// TIA Portal V15.1 export
// export: Created 2024-05-17T05:38:57.2674434Z, ExportSetting WithDefaults, DisplayName Totally Integrated Automation Portal, DisplayVersion V15.1 Update 5, DisplayName TIA Portal Openness, DisplayVersion V15.1 Update 5, DisplayName SINAMICS Startdrive Advanced, DisplayVersion V15.1, DisplayName G130, G150, S120, S150, SINAMICS MV, S210, DisplayVersion V15.1, DisplayName G110M, G120, G120C, G120D, G120P, DisplayVersion V15.1, DisplayName STEP 7 Professional, DisplayVersion V15.1 Update 5, DisplayName STEP 7 Safety, DisplayVersion V15.1, DisplayName WinCC Professional, DisplayVersion V15.1 Update 5, DisplayName SIMATIC Visualization Architect, DisplayVersion V15.1
FUNCTION "209210ZS01PNIODiag" : Void   // FC324, FBD
TITLE = 209210ZS01PNIODiag
{ S7_Optimized_Access := 'FALSE' }
AUTHOR : JS
NAME : Mot001
VERSION : 0.1
// stored: AutoNumber false, IsIECCheckEnabled false, SetENOAutomatically False, UDAEnableTagReadback false
   VAR_OUTPUT
      O_AlarmA : Bool;   // Alarm A
      O_AlarmB : Bool;   // Alarm B
      O_AlarmC : Bool;   // Alarm C
      O_AlarmD : Bool;   // Alarm D
      O_AlarmABCondition : Bool;   // Alarms resetable
      H_IAnim : Word;   // Animation bits to Icon in WinCC
   END_VAR
   VAR_TEMP   // added for the SCL form of the ladder/FBD networks
      _w1 : Bool;
   END_VAR
BEGIN

REGION Network 1: **** --------------------- ET200sp I/O --------------------- ****
END_REGION

REGION Network 2: **** 3 - Communication - Devices **** 209210AS10-JW40 - ET200sp I/O - Busnode 210AS10 - node 40
   // Profinet device don't exist - ET200sp I/O - Busnode 210AS10 - node 40
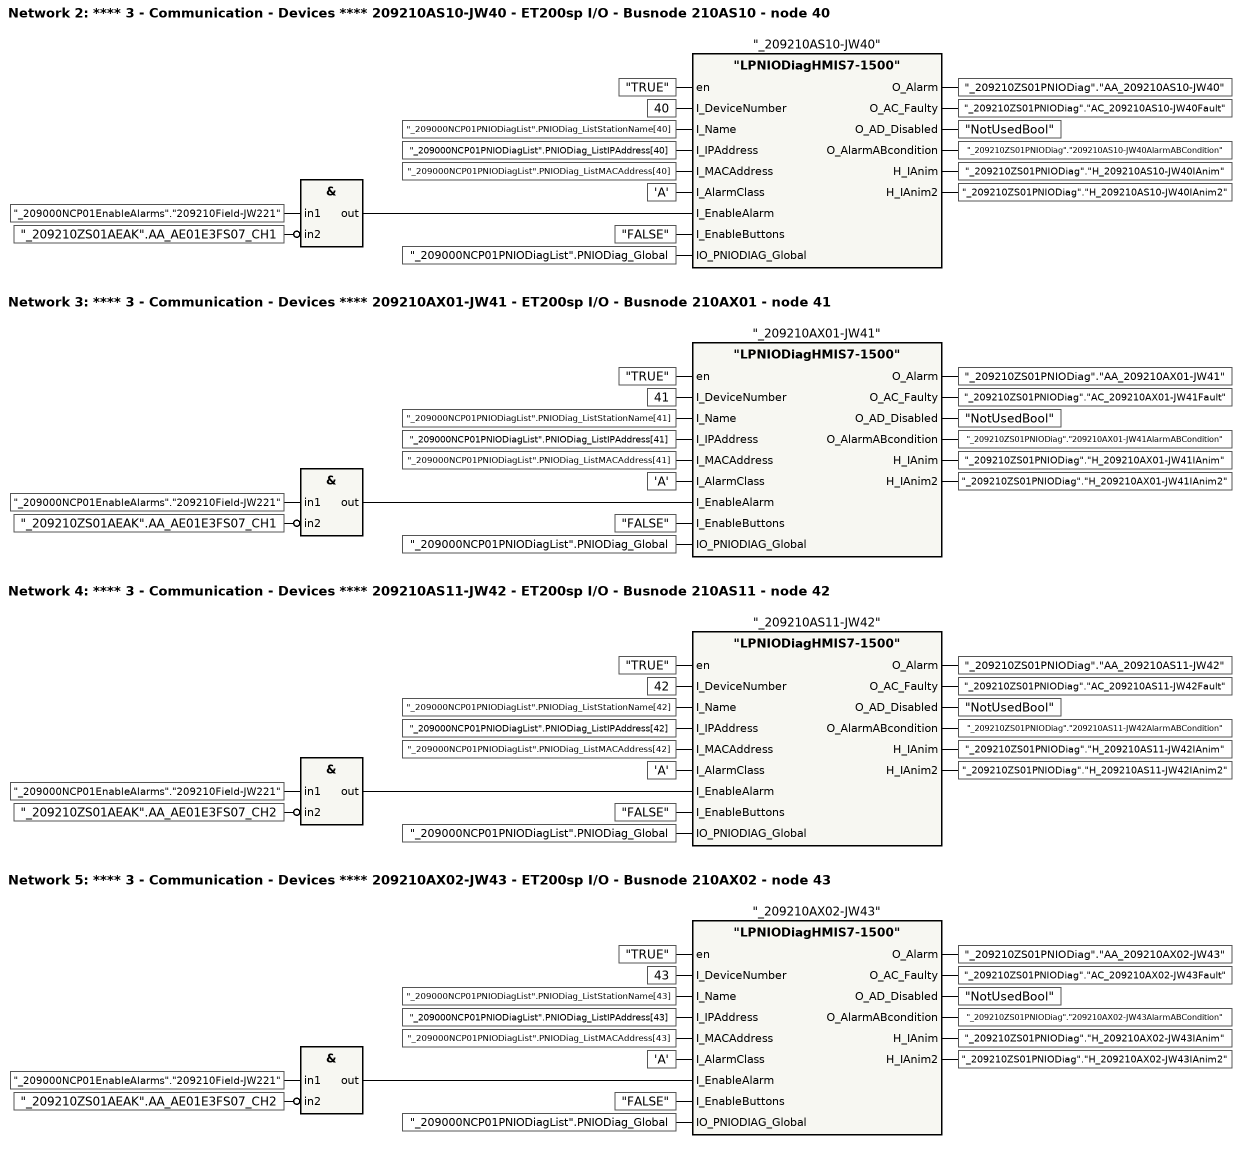
   IF "TRUE" THEN
       "_209210AS10-JW40"(I_DeviceNumber := 40,   // "LPNIODiagHMIS7-1500"
                          I_Name := "_209000NCP01PNIODiagList".PNIODiag_ListStationName[40],
                          I_IPAddress := "_209000NCP01PNIODiagList".PNIODiag_ListIPAddress[40],
                          I_MACAddress := "_209000NCP01PNIODiagList".PNIODiag_ListMACAddress[40],
                          I_AlarmClass := 'A',
                          I_EnableAlarm := "_209000NCP01EnableAlarms"."209210Field-JW221" AND NOT "_209210ZS01AEAK".AA_AE01E3FS07_CH1,
                          I_EnableButtons := "FALSE",
                          IO_PNIODIAG_Global := "_209000NCP01PNIODiagList".PNIODiag_Global,
                          O_Alarm => "_209210ZS01PNIODiag"."AA_209210AS10-JW40",
                          O_AC_Faulty => "_209210ZS01PNIODiag"."AC_209210AS10-JW40Fault",
                          O_AD_Disabled => "NotUsedBool",
                          O_AlarmABcondition => "_209210ZS01PNIODiag"."209210AS10-JW40AlarmABCondition",
                          H_IAnim => "_209210ZS01PNIODiag"."H_209210AS10-JW40IAnim",
                          H_IAnim2 => "_209210ZS01PNIODiag"."H_209210AS10-JW40IAnim2");
   END_IF;
END_REGION

REGION Network 3: **** 3 - Communication - Devices **** 209210AX01-JW41 - ET200sp I/O - Busnode 210AX01 - node 41
   // Profinet device don't exist - ET200sp I/O - Busnode 210AX01 - node 41
   IF "TRUE" THEN
       "_209210AX01-JW41"(I_DeviceNumber := 41,   // "LPNIODiagHMIS7-1500"
                          I_Name := "_209000NCP01PNIODiagList".PNIODiag_ListStationName[41],
                          I_IPAddress := "_209000NCP01PNIODiagList".PNIODiag_ListIPAddress[41],
                          I_MACAddress := "_209000NCP01PNIODiagList".PNIODiag_ListMACAddress[41],
                          I_AlarmClass := 'A',
                          I_EnableAlarm := "_209000NCP01EnableAlarms"."209210Field-JW221" AND NOT "_209210ZS01AEAK".AA_AE01E3FS07_CH1,
                          I_EnableButtons := "FALSE",
                          IO_PNIODIAG_Global := "_209000NCP01PNIODiagList".PNIODiag_Global,
                          O_Alarm => "_209210ZS01PNIODiag"."AA_209210AX01-JW41",
                          O_AC_Faulty => "_209210ZS01PNIODiag"."AC_209210AX01-JW41Fault",
                          O_AD_Disabled => "NotUsedBool",
                          O_AlarmABcondition => "_209210ZS01PNIODiag"."209210AX01-JW41AlarmABCondition",
                          H_IAnim => "_209210ZS01PNIODiag"."H_209210AX01-JW41IAnim",
                          H_IAnim2 => "_209210ZS01PNIODiag"."H_209210AX01-JW41IAnim2");
   END_IF;
END_REGION

REGION Network 4: **** 3 - Communication - Devices **** 209210AS11-JW42 - ET200sp I/O - Busnode 210AS11 - node 42
   // Profinet device don't exist - ET200sp I/O - Busnode 210AS11 - node 42
   IF "TRUE" THEN
       "_209210AS11-JW42"(I_DeviceNumber := 42,   // "LPNIODiagHMIS7-1500"
                          I_Name := "_209000NCP01PNIODiagList".PNIODiag_ListStationName[42],
                          I_IPAddress := "_209000NCP01PNIODiagList".PNIODiag_ListIPAddress[42],
                          I_MACAddress := "_209000NCP01PNIODiagList".PNIODiag_ListMACAddress[42],
                          I_AlarmClass := 'A',
                          I_EnableAlarm := "_209000NCP01EnableAlarms"."209210Field-JW221" AND NOT "_209210ZS01AEAK".AA_AE01E3FS07_CH2,
                          I_EnableButtons := "FALSE",
                          IO_PNIODIAG_Global := "_209000NCP01PNIODiagList".PNIODiag_Global,
                          O_Alarm => "_209210ZS01PNIODiag"."AA_209210AS11-JW42",
                          O_AC_Faulty => "_209210ZS01PNIODiag"."AC_209210AS11-JW42Fault",
                          O_AD_Disabled => "NotUsedBool",
                          O_AlarmABcondition => "_209210ZS01PNIODiag"."209210AS11-JW42AlarmABCondition",
                          H_IAnim => "_209210ZS01PNIODiag"."H_209210AS11-JW42IAnim",
                          H_IAnim2 => "_209210ZS01PNIODiag"."H_209210AS11-JW42IAnim2");
   END_IF;
END_REGION

REGION Network 5: **** 3 - Communication - Devices **** 209210AX02-JW43 - ET200sp I/O - Busnode 210AX02 - node 43
   // Profinet device don't exist - ET200sp I/O - Busnode 210AX02 - node 43
   IF "TRUE" THEN
       "_209210AX02-JW43"(I_DeviceNumber := 43,   // "LPNIODiagHMIS7-1500"
                          I_Name := "_209000NCP01PNIODiagList".PNIODiag_ListStationName[43],
                          I_IPAddress := "_209000NCP01PNIODiagList".PNIODiag_ListIPAddress[43],
                          I_MACAddress := "_209000NCP01PNIODiagList".PNIODiag_ListMACAddress[43],
                          I_AlarmClass := 'A',
                          I_EnableAlarm := "_209000NCP01EnableAlarms"."209210Field-JW221" AND NOT "_209210ZS01AEAK".AA_AE01E3FS07_CH2,
                          I_EnableButtons := "FALSE",
                          IO_PNIODIAG_Global := "_209000NCP01PNIODiagList".PNIODiag_Global,
                          O_Alarm => "_209210ZS01PNIODiag"."AA_209210AX02-JW43",
                          O_AC_Faulty => "_209210ZS01PNIODiag"."AC_209210AX02-JW43Fault",
                          O_AD_Disabled => "NotUsedBool",
                          O_AlarmABcondition => "_209210ZS01PNIODiag"."209210AX02-JW43AlarmABCondition",
                          H_IAnim => "_209210ZS01PNIODiag"."H_209210AX02-JW43IAnim",
                          H_IAnim2 => "_209210ZS01PNIODiag"."H_209210AX02-JW43IAnim2");
   END_IF;
END_REGION

REGION Network 6: **** 3 - Communication - Devices **** 209210AS20-JW48 - ET200sp I/O - Busnode 210AS20 - node 48
   // Profinet device don't exist - ET200sp I/O - Busnode 210AS20 - node 48
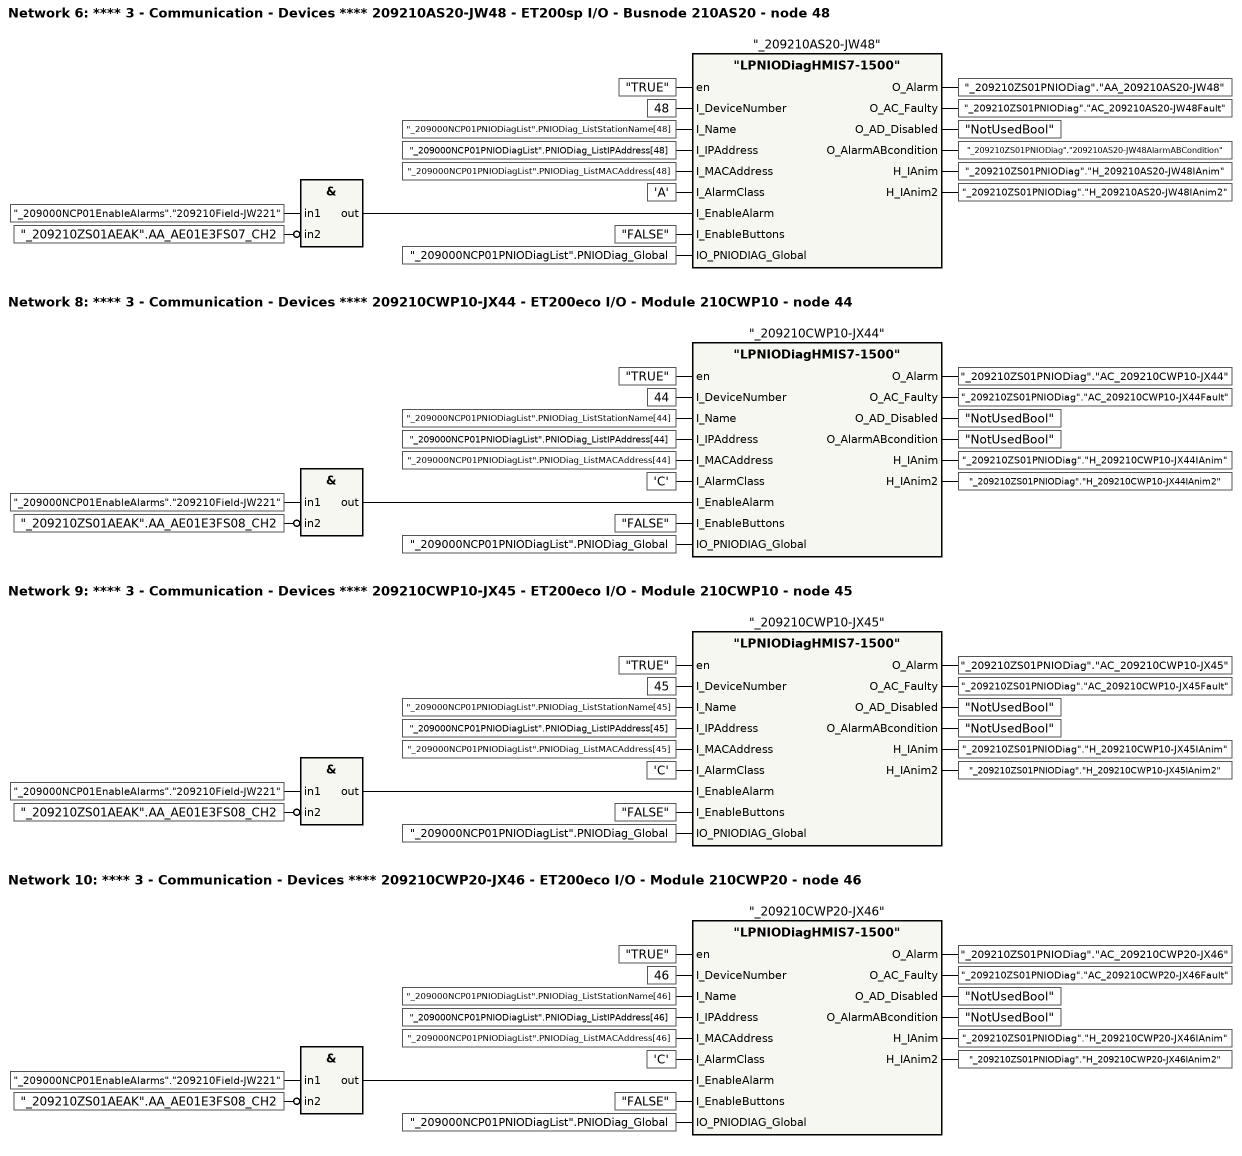
   IF "TRUE" THEN
       "_209210AS20-JW48"(I_DeviceNumber := 48,   // "LPNIODiagHMIS7-1500"
                          I_Name := "_209000NCP01PNIODiagList".PNIODiag_ListStationName[48],
                          I_IPAddress := "_209000NCP01PNIODiagList".PNIODiag_ListIPAddress[48],
                          I_MACAddress := "_209000NCP01PNIODiagList".PNIODiag_ListMACAddress[48],
                          I_AlarmClass := 'A',
                          I_EnableAlarm := "_209000NCP01EnableAlarms"."209210Field-JW221" AND NOT "_209210ZS01AEAK".AA_AE01E3FS07_CH2,
                          I_EnableButtons := "FALSE",
                          IO_PNIODIAG_Global := "_209000NCP01PNIODiagList".PNIODiag_Global,
                          O_Alarm => "_209210ZS01PNIODiag"."AA_209210AS20-JW48",
                          O_AC_Faulty => "_209210ZS01PNIODiag"."AC_209210AS20-JW48Fault",
                          O_AD_Disabled => "NotUsedBool",
                          O_AlarmABcondition => "_209210ZS01PNIODiag"."209210AS20-JW48AlarmABCondition",
                          H_IAnim => "_209210ZS01PNIODiag"."H_209210AS20-JW48IAnim",
                          H_IAnim2 => "_209210ZS01PNIODiag"."H_209210AS20-JW48IAnim2");
   END_IF;
END_REGION

REGION Network 7: **** --------------------- ET200eco I/O --------------------- ****
END_REGION

REGION Network 8: **** 3 - Communication - Devices **** 209210CWP10-JX44 - ET200eco I/O - Module 210CWP10 - node 44
   // Profinet device don't exist - ET200eco I/O - Module 210CWP10 - node 44
   IF "TRUE" THEN
       "_209210CWP10-JX44"(I_DeviceNumber := 44,   // "LPNIODiagHMIS7-1500"
                           I_Name := "_209000NCP01PNIODiagList".PNIODiag_ListStationName[44],
                           I_IPAddress := "_209000NCP01PNIODiagList".PNIODiag_ListIPAddress[44],
                           I_MACAddress := "_209000NCP01PNIODiagList".PNIODiag_ListMACAddress[44],
                           I_AlarmClass := 'C',
                           I_EnableAlarm := "_209000NCP01EnableAlarms"."209210Field-JW221" AND NOT "_209210ZS01AEAK".AA_AE01E3FS08_CH2,
                           I_EnableButtons := "FALSE",
                           IO_PNIODIAG_Global := "_209000NCP01PNIODiagList".PNIODiag_Global,
                           O_Alarm => "_209210ZS01PNIODiag"."AC_209210CWP10-JX44",
                           O_AC_Faulty => "_209210ZS01PNIODiag"."AC_209210CWP10-JX44Fault",
                           O_AD_Disabled => "NotUsedBool",
                           O_AlarmABcondition => "NotUsedBool",
                           H_IAnim => "_209210ZS01PNIODiag"."H_209210CWP10-JX44IAnim",
                           H_IAnim2 => "_209210ZS01PNIODiag"."H_209210CWP10-JX44IAnim2");
   END_IF;
END_REGION

REGION Network 9: **** 3 - Communication - Devices **** 209210CWP10-JX45 - ET200eco I/O - Module 210CWP10 - node 45
   // Profinet device don't exist - ET200eco I/O - Module 210CWP10 - node 45
   IF "TRUE" THEN
       "_209210CWP10-JX45"(I_DeviceNumber := 45,   // "LPNIODiagHMIS7-1500"
                           I_Name := "_209000NCP01PNIODiagList".PNIODiag_ListStationName[45],
                           I_IPAddress := "_209000NCP01PNIODiagList".PNIODiag_ListIPAddress[45],
                           I_MACAddress := "_209000NCP01PNIODiagList".PNIODiag_ListMACAddress[45],
                           I_AlarmClass := 'C',
                           I_EnableAlarm := "_209000NCP01EnableAlarms"."209210Field-JW221" AND NOT "_209210ZS01AEAK".AA_AE01E3FS08_CH2,
                           I_EnableButtons := "FALSE",
                           IO_PNIODIAG_Global := "_209000NCP01PNIODiagList".PNIODiag_Global,
                           O_Alarm => "_209210ZS01PNIODiag"."AC_209210CWP10-JX45",
                           O_AC_Faulty => "_209210ZS01PNIODiag"."AC_209210CWP10-JX45Fault",
                           O_AD_Disabled => "NotUsedBool",
                           O_AlarmABcondition => "NotUsedBool",
                           H_IAnim => "_209210ZS01PNIODiag"."H_209210CWP10-JX45IAnim",
                           H_IAnim2 => "_209210ZS01PNIODiag"."H_209210CWP10-JX45IAnim2");
   END_IF;
END_REGION

REGION Network 10: **** 3 - Communication - Devices **** 209210CWP20-JX46 - ET200eco I/O - Module 210CWP20 - node 46
   // Profinet device don't exist - ET200eco I/O - Module 210CWP20 - node 46
   IF "TRUE" THEN
       "_209210CWP20-JX46"(I_DeviceNumber := 46,   // "LPNIODiagHMIS7-1500"
                           I_Name := "_209000NCP01PNIODiagList".PNIODiag_ListStationName[46],
                           I_IPAddress := "_209000NCP01PNIODiagList".PNIODiag_ListIPAddress[46],
                           I_MACAddress := "_209000NCP01PNIODiagList".PNIODiag_ListMACAddress[46],
                           I_AlarmClass := 'C',
                           I_EnableAlarm := "_209000NCP01EnableAlarms"."209210Field-JW221" AND NOT "_209210ZS01AEAK".AA_AE01E3FS08_CH2,
                           I_EnableButtons := "FALSE",
                           IO_PNIODIAG_Global := "_209000NCP01PNIODiagList".PNIODiag_Global,
                           O_Alarm => "_209210ZS01PNIODiag"."AC_209210CWP20-JX46",
                           O_AC_Faulty => "_209210ZS01PNIODiag"."AC_209210CWP20-JX46Fault",
                           O_AD_Disabled => "NotUsedBool",
                           O_AlarmABcondition => "NotUsedBool",
                           H_IAnim => "_209210ZS01PNIODiag"."H_209210CWP20-JX46IAnim",
                           H_IAnim2 => "_209210ZS01PNIODiag"."H_209210CWP20-JX46IAnim2");
   END_IF;
END_REGION

REGION Network 11: **** 3 - Communication - Devices **** 209210CWP20-JX47 - ET200eco I/O - Module 210CWP20 - node 47
   // Profinet device don't exist - ET200eco I/O - Module 210CWP20 - node 47
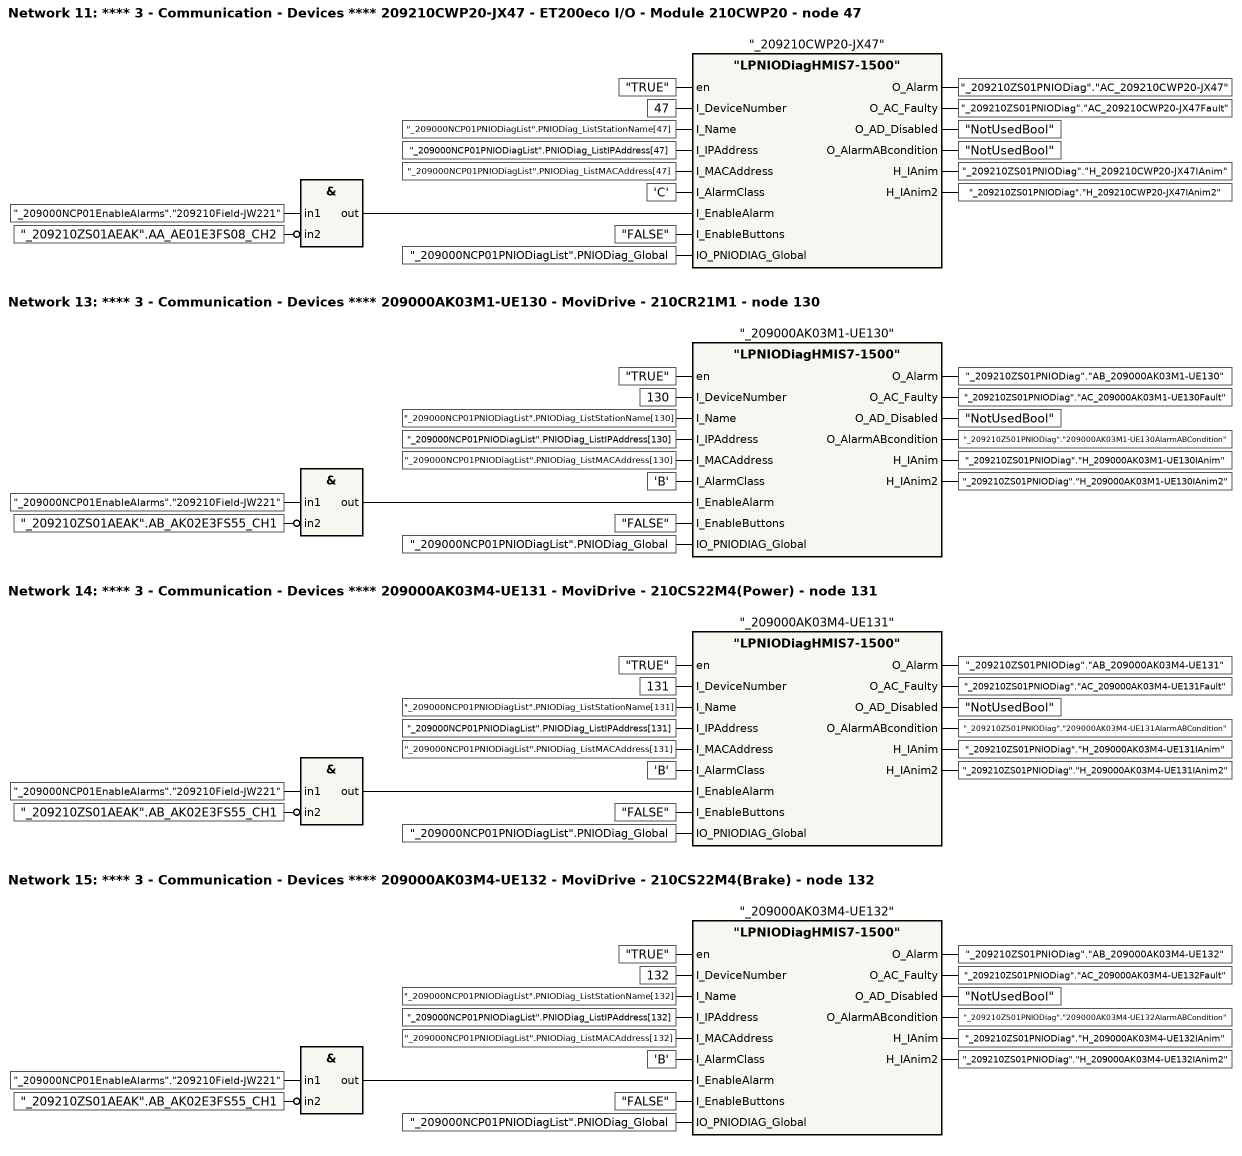
   IF "TRUE" THEN
       "_209210CWP20-JX47"(I_DeviceNumber := 47,   // "LPNIODiagHMIS7-1500"
                           I_Name := "_209000NCP01PNIODiagList".PNIODiag_ListStationName[47],
                           I_IPAddress := "_209000NCP01PNIODiagList".PNIODiag_ListIPAddress[47],
                           I_MACAddress := "_209000NCP01PNIODiagList".PNIODiag_ListMACAddress[47],
                           I_AlarmClass := 'C',
                           I_EnableAlarm := "_209000NCP01EnableAlarms"."209210Field-JW221" AND NOT "_209210ZS01AEAK".AA_AE01E3FS08_CH2,
                           I_EnableButtons := "FALSE",
                           IO_PNIODIAG_Global := "_209000NCP01PNIODiagList".PNIODiag_Global,
                           O_Alarm => "_209210ZS01PNIODiag"."AC_209210CWP20-JX47",
                           O_AC_Faulty => "_209210ZS01PNIODiag"."AC_209210CWP20-JX47Fault",
                           O_AD_Disabled => "NotUsedBool",
                           O_AlarmABcondition => "NotUsedBool",
                           H_IAnim => "_209210ZS01PNIODiag"."H_209210CWP20-JX47IAnim",
                           H_IAnim2 => "_209210ZS01PNIODiag"."H_209210CWP20-JX47IAnim2");
   END_IF;
END_REGION

REGION Network 12: **** --------------------- Drive --------------------- ****
END_REGION

REGION Network 13: **** 3 - Communication - Devices **** 209000AK03M1-UE130 - MoviDrive - 210CR21M1 - node 130
   // Profinet device don't exist - MoviDrive - 210CR21M1 - node 130
   IF "TRUE" THEN
       "_209000AK03M1-UE130"(I_DeviceNumber := 130,   // "LPNIODiagHMIS7-1500"
                             I_Name := "_209000NCP01PNIODiagList".PNIODiag_ListStationName[130],
                             I_IPAddress := "_209000NCP01PNIODiagList".PNIODiag_ListIPAddress[130],
                             I_MACAddress := "_209000NCP01PNIODiagList".PNIODiag_ListMACAddress[130],
                             I_AlarmClass := 'B',
                             I_EnableAlarm := "_209000NCP01EnableAlarms"."209210Field-JW221" AND NOT "_209210ZS01AEAK".AB_AK02E3FS55_CH1,
                             I_EnableButtons := "FALSE",
                             IO_PNIODIAG_Global := "_209000NCP01PNIODiagList".PNIODiag_Global,
                             O_Alarm => "_209210ZS01PNIODiag"."AB_209000AK03M1-UE130",
                             O_AC_Faulty => "_209210ZS01PNIODiag"."AC_209000AK03M1-UE130Fault",
                             O_AD_Disabled => "NotUsedBool",
                             O_AlarmABcondition => "_209210ZS01PNIODiag"."209000AK03M1-UE130AlarmABCondition",
                             H_IAnim => "_209210ZS01PNIODiag"."H_209000AK03M1-UE130IAnim",
                             H_IAnim2 => "_209210ZS01PNIODiag"."H_209000AK03M1-UE130IAnim2");
   END_IF;
END_REGION

REGION Network 14: **** 3 - Communication - Devices **** 209000AK03M4-UE131 - MoviDrive - 210CS22M4(Power) - node 131
   // Profinet device don't exist - MoviDrive - 210CS22M4(Power) - node 131
   IF "TRUE" THEN
       "_209000AK03M4-UE131"(I_DeviceNumber := 131,   // "LPNIODiagHMIS7-1500"
                             I_Name := "_209000NCP01PNIODiagList".PNIODiag_ListStationName[131],
                             I_IPAddress := "_209000NCP01PNIODiagList".PNIODiag_ListIPAddress[131],
                             I_MACAddress := "_209000NCP01PNIODiagList".PNIODiag_ListMACAddress[131],
                             I_AlarmClass := 'B',
                             I_EnableAlarm := "_209000NCP01EnableAlarms"."209210Field-JW221" AND NOT "_209210ZS01AEAK".AB_AK02E3FS55_CH1,
                             I_EnableButtons := "FALSE",
                             IO_PNIODIAG_Global := "_209000NCP01PNIODiagList".PNIODiag_Global,
                             O_Alarm => "_209210ZS01PNIODiag"."AB_209000AK03M4-UE131",
                             O_AC_Faulty => "_209210ZS01PNIODiag"."AC_209000AK03M4-UE131Fault",
                             O_AD_Disabled => "NotUsedBool",
                             O_AlarmABcondition => "_209210ZS01PNIODiag"."209000AK03M4-UE131AlarmABCondition",
                             H_IAnim => "_209210ZS01PNIODiag"."H_209000AK03M4-UE131IAnim",
                             H_IAnim2 => "_209210ZS01PNIODiag"."H_209000AK03M4-UE131IAnim2");
   END_IF;
END_REGION

REGION Network 15: **** 3 - Communication - Devices **** 209000AK03M4-UE132 - MoviDrive - 210CS22M4(Brake) - node 132
   // Profinet device don't exist - MoviDrive - 210CS22M4(Brake) - node 132
   IF "TRUE" THEN
       "_209000AK03M4-UE132"(I_DeviceNumber := 132,   // "LPNIODiagHMIS7-1500"
                             I_Name := "_209000NCP01PNIODiagList".PNIODiag_ListStationName[132],
                             I_IPAddress := "_209000NCP01PNIODiagList".PNIODiag_ListIPAddress[132],
                             I_MACAddress := "_209000NCP01PNIODiagList".PNIODiag_ListMACAddress[132],
                             I_AlarmClass := 'B',
                             I_EnableAlarm := "_209000NCP01EnableAlarms"."209210Field-JW221" AND NOT "_209210ZS01AEAK".AB_AK02E3FS55_CH1,
                             I_EnableButtons := "FALSE",
                             IO_PNIODIAG_Global := "_209000NCP01PNIODiagList".PNIODiag_Global,
                             O_Alarm => "_209210ZS01PNIODiag"."AB_209000AK03M4-UE132",
                             O_AC_Faulty => "_209210ZS01PNIODiag"."AC_209000AK03M4-UE132Fault",
                             O_AD_Disabled => "NotUsedBool",
                             O_AlarmABcondition => "_209210ZS01PNIODiag"."209000AK03M4-UE132AlarmABCondition",
                             H_IAnim => "_209210ZS01PNIODiag"."H_209000AK03M4-UE132IAnim",
                             H_IAnim2 => "_209210ZS01PNIODiag"."H_209000AK03M4-UE132IAnim2");
   END_IF;
END_REGION

REGION Network 16: **** 3 - Communication - Devices **** 209000AK03M1-UE133 - MoviDrive - 210CR23M1 - node 133
   // Profinet device don't exist - MoviDrive - 210CR23M1 - node 133
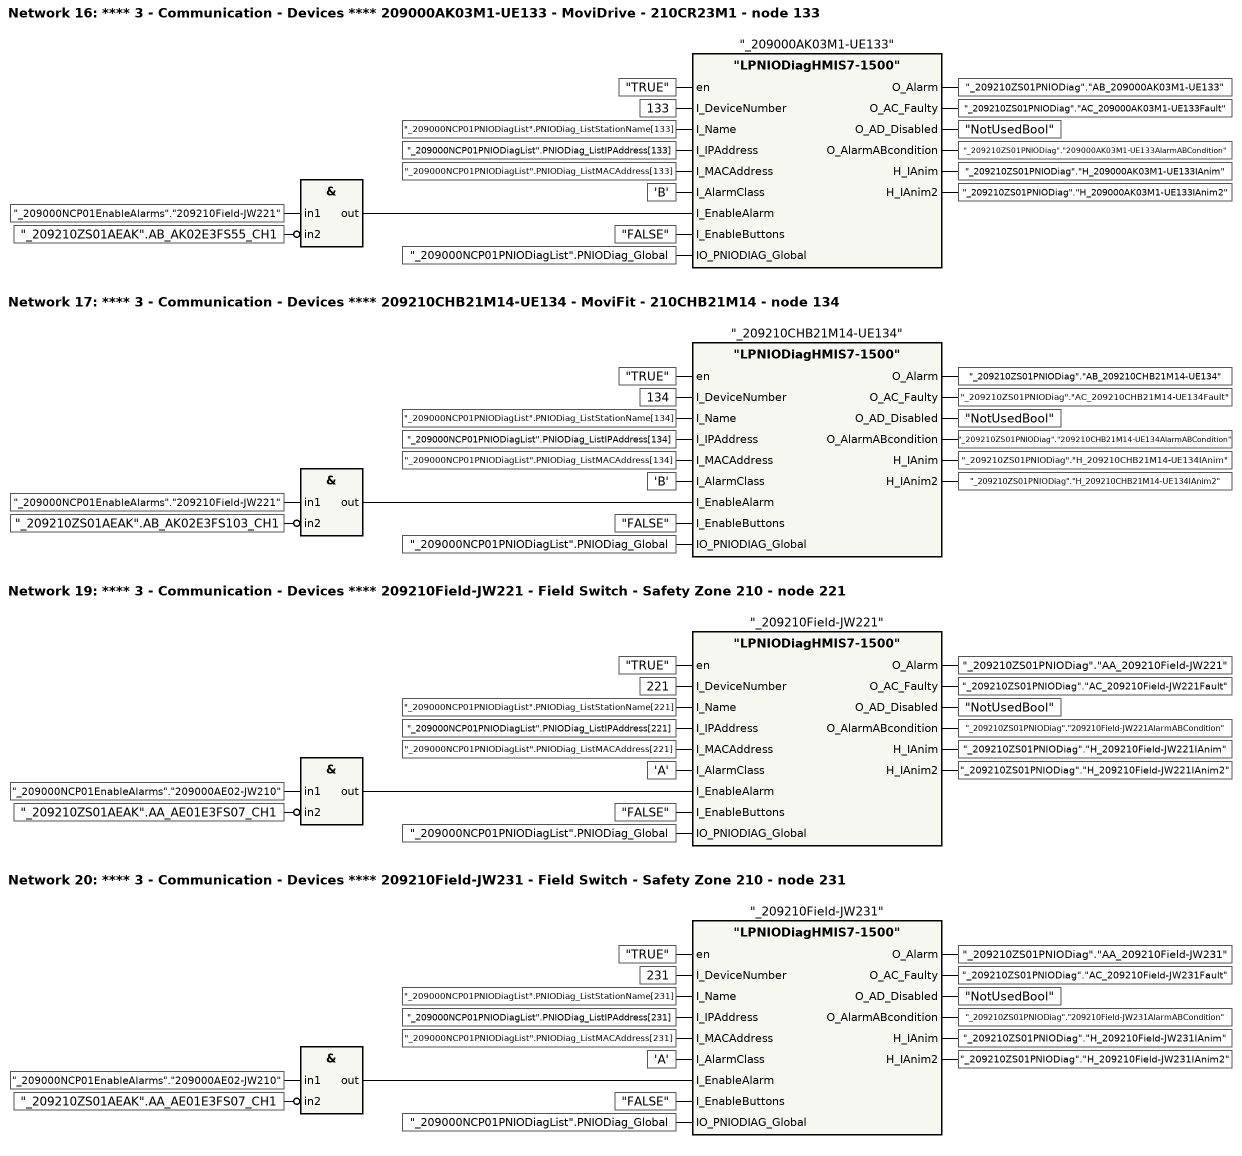
   IF "TRUE" THEN
       "_209000AK03M1-UE133"(I_DeviceNumber := 133,   // "LPNIODiagHMIS7-1500"
                             I_Name := "_209000NCP01PNIODiagList".PNIODiag_ListStationName[133],
                             I_IPAddress := "_209000NCP01PNIODiagList".PNIODiag_ListIPAddress[133],
                             I_MACAddress := "_209000NCP01PNIODiagList".PNIODiag_ListMACAddress[133],
                             I_AlarmClass := 'B',
                             I_EnableAlarm := "_209000NCP01EnableAlarms"."209210Field-JW221" AND NOT "_209210ZS01AEAK".AB_AK02E3FS55_CH1,
                             I_EnableButtons := "FALSE",
                             IO_PNIODIAG_Global := "_209000NCP01PNIODiagList".PNIODiag_Global,
                             O_Alarm => "_209210ZS01PNIODiag"."AB_209000AK03M1-UE133",
                             O_AC_Faulty => "_209210ZS01PNIODiag"."AC_209000AK03M1-UE133Fault",
                             O_AD_Disabled => "NotUsedBool",
                             O_AlarmABcondition => "_209210ZS01PNIODiag"."209000AK03M1-UE133AlarmABCondition",
                             H_IAnim => "_209210ZS01PNIODiag"."H_209000AK03M1-UE133IAnim",
                             H_IAnim2 => "_209210ZS01PNIODiag"."H_209000AK03M1-UE133IAnim2");
   END_IF;
END_REGION

REGION Network 17: **** 3 - Communication - Devices **** 209210CHB21M14-UE134 - MoviFit - 210CHB21M14 - node 134
   // Profinet device don't exist - MoviFit - 210CHB21M14 - node 134
   IF "TRUE" THEN
       "_209210CHB21M14-UE134"(I_DeviceNumber := 134,   // "LPNIODiagHMIS7-1500"
                               I_Name := "_209000NCP01PNIODiagList".PNIODiag_ListStationName[134],
                               I_IPAddress := "_209000NCP01PNIODiagList".PNIODiag_ListIPAddress[134],
                               I_MACAddress := "_209000NCP01PNIODiagList".PNIODiag_ListMACAddress[134],
                               I_AlarmClass := 'B',
                               I_EnableAlarm := "_209000NCP01EnableAlarms"."209210Field-JW221" AND NOT "_209210ZS01AEAK".AB_AK02E3FS103_CH1,
                               I_EnableButtons := "FALSE",
                               IO_PNIODIAG_Global := "_209000NCP01PNIODiagList".PNIODiag_Global,
                               O_Alarm => "_209210ZS01PNIODiag"."AB_209210CHB21M14-UE134",
                               O_AC_Faulty => "_209210ZS01PNIODiag"."AC_209210CHB21M14-UE134Fault",
                               O_AD_Disabled => "NotUsedBool",
                               O_AlarmABcondition => "_209210ZS01PNIODiag"."209210CHB21M14-UE134AlarmABCondition",
                               H_IAnim => "_209210ZS01PNIODiag"."H_209210CHB21M14-UE134IAnim",
                               H_IAnim2 => "_209210ZS01PNIODiag"."H_209210CHB21M14-UE134IAnim2");
   END_IF;
END_REGION

REGION Network 18: **** --------------------- Field Switch --------------------- ****
END_REGION

REGION Network 19: **** 3 - Communication - Devices **** 209210Field-JW221 - Field Switch - Safety Zone 210 - node 221
   // Profinet device don't exist - Field Switch - Safety Zone 210 - node 221
   IF "TRUE" THEN
       "_209210Field-JW221"(I_DeviceNumber := 221,   // "LPNIODiagHMIS7-1500"
                            I_Name := "_209000NCP01PNIODiagList".PNIODiag_ListStationName[221],
                            I_IPAddress := "_209000NCP01PNIODiagList".PNIODiag_ListIPAddress[221],
                            I_MACAddress := "_209000NCP01PNIODiagList".PNIODiag_ListMACAddress[221],
                            I_AlarmClass := 'A',
                            I_EnableAlarm := "_209000NCP01EnableAlarms"."209000AE02-JW210" AND NOT "_209210ZS01AEAK".AA_AE01E3FS07_CH1,
                            I_EnableButtons := "FALSE",
                            IO_PNIODIAG_Global := "_209000NCP01PNIODiagList".PNIODiag_Global,
                            O_Alarm => "_209210ZS01PNIODiag"."AA_209210Field-JW221",
                            O_AC_Faulty => "_209210ZS01PNIODiag"."AC_209210Field-JW221Fault",
                            O_AD_Disabled => "NotUsedBool",
                            O_AlarmABcondition => "_209210ZS01PNIODiag"."209210Field-JW221AlarmABCondition",
                            H_IAnim => "_209210ZS01PNIODiag"."H_209210Field-JW221IAnim",
                            H_IAnim2 => "_209210ZS01PNIODiag"."H_209210Field-JW221IAnim2");
   END_IF;
END_REGION

REGION Network 20: **** 3 - Communication - Devices **** 209210Field-JW231 - Field Switch - Safety Zone 210 - node 231
   // Profinet device don't exist - Field Switch - Safety Zone 210 - node 231
   IF "TRUE" THEN
       "_209210Field-JW231"(I_DeviceNumber := 231,   // "LPNIODiagHMIS7-1500"
                            I_Name := "_209000NCP01PNIODiagList".PNIODiag_ListStationName[231],
                            I_IPAddress := "_209000NCP01PNIODiagList".PNIODiag_ListIPAddress[231],
                            I_MACAddress := "_209000NCP01PNIODiagList".PNIODiag_ListMACAddress[231],
                            I_AlarmClass := 'A',
                            I_EnableAlarm := "_209000NCP01EnableAlarms"."209000AE02-JW210" AND NOT "_209210ZS01AEAK".AA_AE01E3FS07_CH1,
                            I_EnableButtons := "FALSE",
                            IO_PNIODIAG_Global := "_209000NCP01PNIODiagList".PNIODiag_Global,
                            O_Alarm => "_209210ZS01PNIODiag"."AA_209210Field-JW231",
                            O_AC_Faulty => "_209210ZS01PNIODiag"."AC_209210Field-JW231Fault",
                            O_AD_Disabled => "NotUsedBool",
                            O_AlarmABcondition => "_209210ZS01PNIODiag"."209210Field-JW231AlarmABCondition",
                            H_IAnim => "_209210ZS01PNIODiag"."H_209210Field-JW231IAnim",
                            H_IAnim2 => "_209210ZS01PNIODiag"."H_209210Field-JW231IAnim2");
   END_IF;
END_REGION

REGION Network 21: **** -------------------------------------------------- ****
END_REGION

REGION Network 22: **** 4.6 - Machine Status - Indications **** Icon animation
   // Icon animation
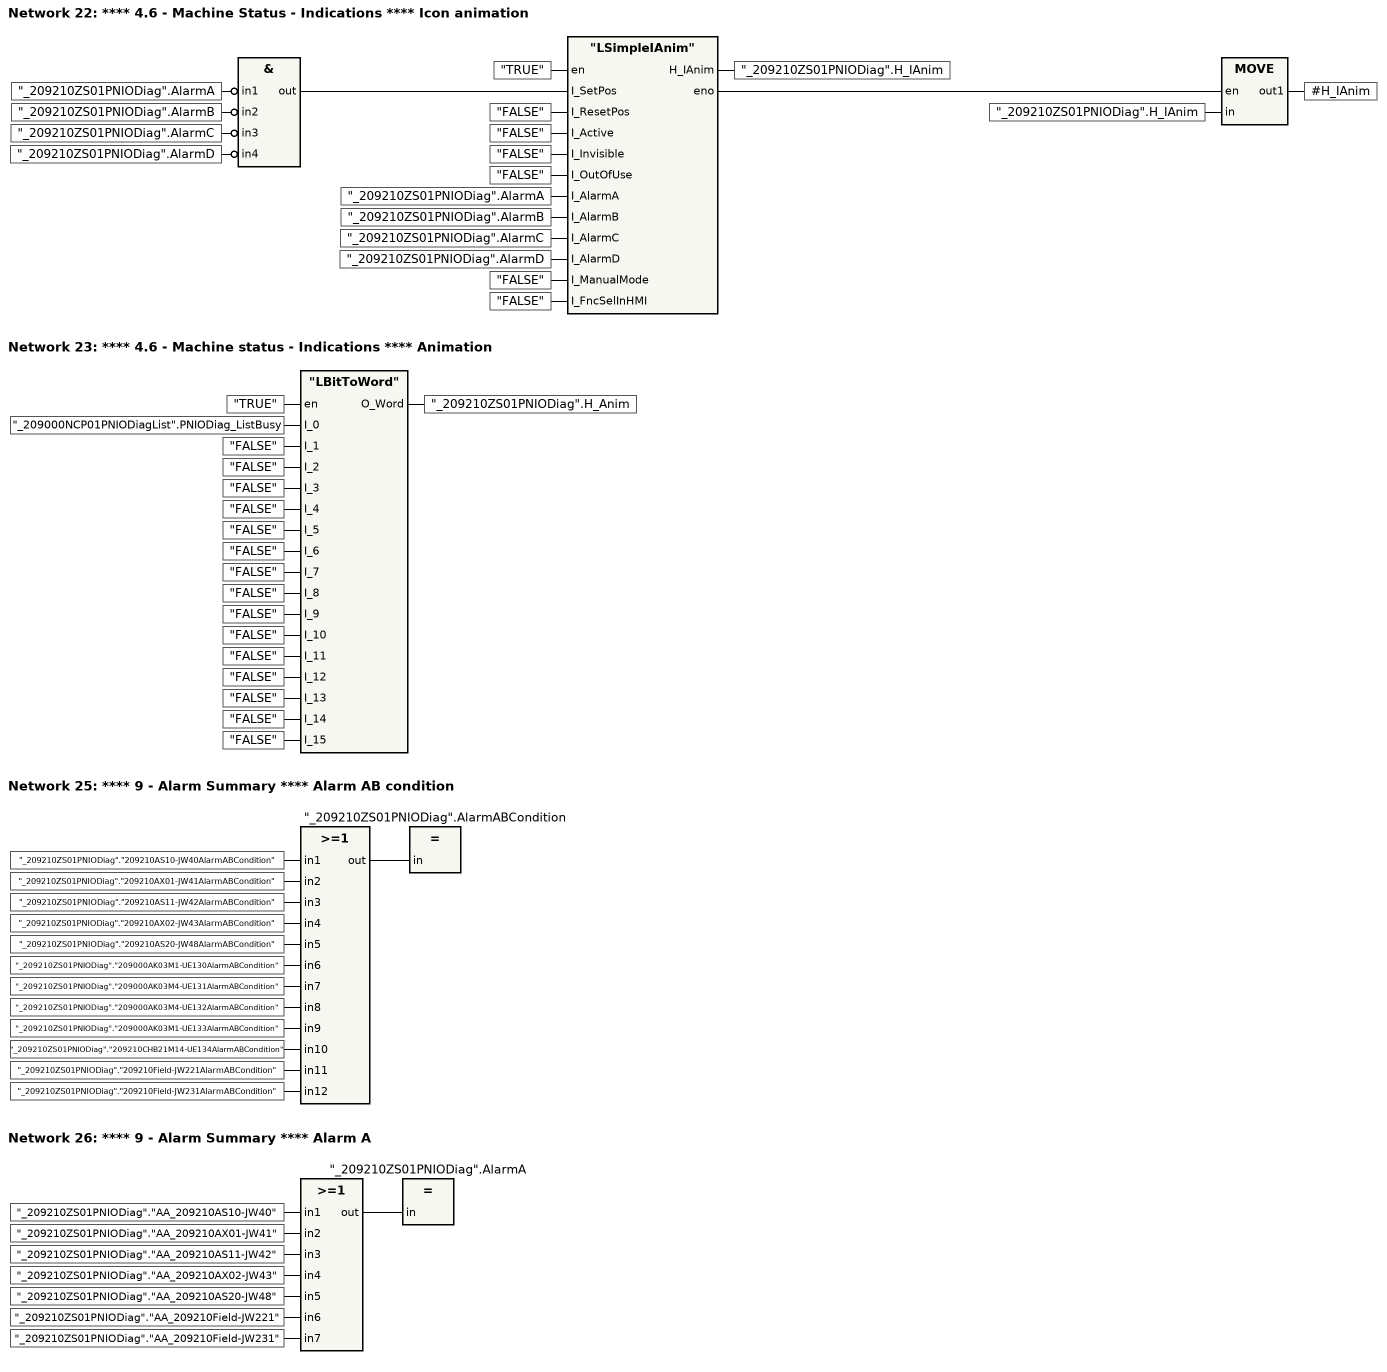
   "LSimpleIAnim"(EN := "TRUE",
                  I_SetPos := NOT "_209210ZS01PNIODiag".AlarmA AND NOT "_209210ZS01PNIODiag".AlarmB AND NOT "_209210ZS01PNIODiag".AlarmC AND NOT "_209210ZS01PNIODiag".AlarmD,
                  I_ResetPos := "FALSE",
                  I_Active := "FALSE",
                  I_Invisible := "FALSE",
                  I_OutOfUse := "FALSE",
                  I_AlarmA := "_209210ZS01PNIODiag".AlarmA,
                  I_AlarmB := "_209210ZS01PNIODiag".AlarmB,
                  I_AlarmC := "_209210ZS01PNIODiag".AlarmC,
                  I_AlarmD := "_209210ZS01PNIODiag".AlarmD,
                  I_ManualMode := "FALSE",
                  I_FncSelInHMI := "FALSE",
                  H_IAnim => "_209210ZS01PNIODiag".H_IAnim,
                  ENO => #_w1);
   IF #_w1 THEN #H_IAnim := "_209210ZS01PNIODiag".H_IAnim; END_IF;
END_REGION

REGION Network 23: **** 4.6 - Machine status - Indications **** Animation
   // Animation
   IF "TRUE" THEN
       "LBitToWord"(I_0 := "_209000NCP01PNIODiagList".PNIODiag_ListBusy,
                    I_1 := "FALSE",
                    I_2 := "FALSE",
                    I_3 := "FALSE",
                    I_4 := "FALSE",
                    I_5 := "FALSE",
                    I_6 := "FALSE",
                    I_7 := "FALSE",
                    I_8 := "FALSE",
                    I_9 := "FALSE",
                    I_10 := "FALSE",
                    I_11 := "FALSE",
                    I_12 := "FALSE",
                    I_13 := "FALSE",
                    I_14 := "FALSE",
                    I_15 := "FALSE",
                    O_Word => "_209210ZS01PNIODiag".H_Anim);
   END_IF;
END_REGION

NETWORK
TITLE = **** 4.6 - Machine Status - Indications **** Animation DB number
// DB number
      OPN   "_209210ZS01PNIODiag";
      L     DBNO;
      T     "_209210ZS01PNIODiag".H_DBnr;

REGION Network 25: **** 9 - Alarm Summary **** Alarm AB condition
   // Summary of Alarm AB condition
   "_209210ZS01PNIODiag".AlarmABCondition := "_209210ZS01PNIODiag"."209210AS10-JW40AlarmABCondition" OR "_209210ZS01PNIODiag"."209210AX01-JW41AlarmABCondition" OR "_209210ZS01PNIODiag"."209210AS11-JW42AlarmABCondition" OR "_209210ZS01PNIODiag"."209210AX02-JW43AlarmABCondition" OR "_209210ZS01PNIODiag"."209210AS20-JW48AlarmABCondition" OR "_209210ZS01PNIODiag"."209000AK03M1-UE130AlarmABCondition" OR "_209210ZS01PNIODiag"."209000AK03M4-UE131AlarmABCondition" OR "_209210ZS01PNIODiag"."209000AK03M4-UE132AlarmABCondition" OR "_209210ZS01PNIODiag"."209000AK03M1-UE133AlarmABCondition" OR "_209210ZS01PNIODiag"."209210CHB21M14-UE134AlarmABCondition" OR "_209210ZS01PNIODiag"."209210Field-JW221AlarmABCondition" OR "_209210ZS01PNIODiag"."209210Field-JW231AlarmABCondition";
END_REGION

REGION Network 26: **** 9 - Alarm Summary **** Alarm A
   // Summary of alarms A
   "_209210ZS01PNIODiag".AlarmA := "_209210ZS01PNIODiag"."AA_209210AS10-JW40" OR "_209210ZS01PNIODiag"."AA_209210AX01-JW41" OR "_209210ZS01PNIODiag"."AA_209210AS11-JW42" OR "_209210ZS01PNIODiag"."AA_209210AX02-JW43" OR "_209210ZS01PNIODiag"."AA_209210AS20-JW48" OR "_209210ZS01PNIODiag"."AA_209210Field-JW221" OR "_209210ZS01PNIODiag"."AA_209210Field-JW231";
END_REGION

REGION Network 27: **** 9 - Alarm Summary **** Alarm B
   // Summary of alarms B
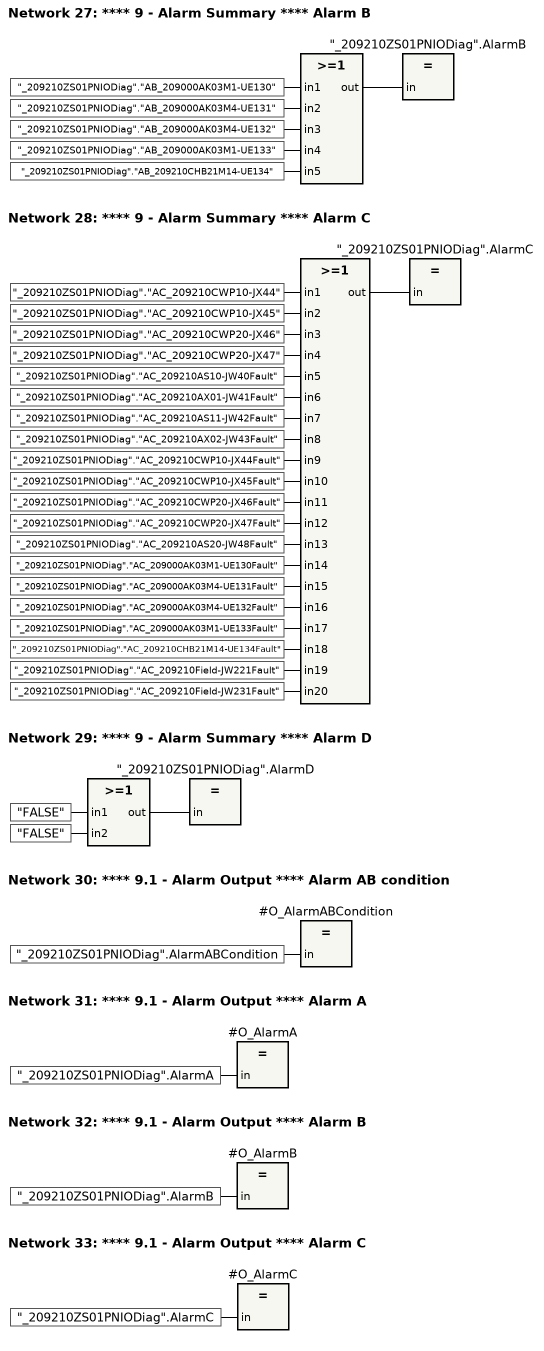
   "_209210ZS01PNIODiag".AlarmB := "_209210ZS01PNIODiag"."AB_209000AK03M1-UE130" OR "_209210ZS01PNIODiag"."AB_209000AK03M4-UE131" OR "_209210ZS01PNIODiag"."AB_209000AK03M4-UE132" OR "_209210ZS01PNIODiag"."AB_209000AK03M1-UE133" OR "_209210ZS01PNIODiag"."AB_209210CHB21M14-UE134";
END_REGION

REGION Network 28: **** 9 - Alarm Summary **** Alarm C
   // Summary of alarms C
   "_209210ZS01PNIODiag".AlarmC := "_209210ZS01PNIODiag"."AC_209210CWP10-JX44" OR "_209210ZS01PNIODiag"."AC_209210CWP10-JX45" OR "_209210ZS01PNIODiag"."AC_209210CWP20-JX46" OR "_209210ZS01PNIODiag"."AC_209210CWP20-JX47" OR "_209210ZS01PNIODiag"."AC_209210AS10-JW40Fault" OR "_209210ZS01PNIODiag"."AC_209210AX01-JW41Fault" OR "_209210ZS01PNIODiag"."AC_209210AS11-JW42Fault" OR "_209210ZS01PNIODiag"."AC_209210AX02-JW43Fault" OR "_209210ZS01PNIODiag"."AC_209210CWP10-JX44Fault" OR "_209210ZS01PNIODiag"."AC_209210CWP10-JX45Fault" OR "_209210ZS01PNIODiag"."AC_209210CWP20-JX46Fault" OR "_209210ZS01PNIODiag"."AC_209210CWP20-JX47Fault" OR "_209210ZS01PNIODiag"."AC_209210AS20-JW48Fault" OR "_209210ZS01PNIODiag"."AC_209000AK03M1-UE130Fault" OR "_209210ZS01PNIODiag"."AC_209000AK03M4-UE131Fault" OR "_209210ZS01PNIODiag"."AC_209000AK03M4-UE132Fault" OR "_209210ZS01PNIODiag"."AC_209000AK03M1-UE133Fault" OR "_209210ZS01PNIODiag"."AC_209210CHB21M14-UE134Fault" OR "_209210ZS01PNIODiag"."AC_209210Field-JW221Fault" OR "_209210ZS01PNIODiag"."AC_209210Field-JW231Fault";
END_REGION

REGION Network 29: **** 9 - Alarm Summary **** Alarm D
   // Summary of alarms D
   "_209210ZS01PNIODiag".AlarmD := "FALSE" OR "FALSE";
END_REGION

REGION Network 30: **** 9.1 - Alarm Output **** Alarm AB condition
   // Alarm AB condition
   #O_AlarmABCondition := "_209210ZS01PNIODiag".AlarmABCondition;
END_REGION

REGION Network 31: **** 9.1 - Alarm Output **** Alarm A
   // Output Alarm A
   #O_AlarmA := "_209210ZS01PNIODiag".AlarmA;
END_REGION

REGION Network 32: **** 9.1 - Alarm Output **** Alarm B
   // Output Alarm B
   #O_AlarmB := "_209210ZS01PNIODiag".AlarmB;
END_REGION

REGION Network 33: **** 9.1 - Alarm Output **** Alarm C
   // Output Alarm A
   #O_AlarmC := "_209210ZS01PNIODiag".AlarmC;
END_REGION

REGION Network 34: **** 9.1 - Alarm Output **** Alarm D
   // Output Alarm D
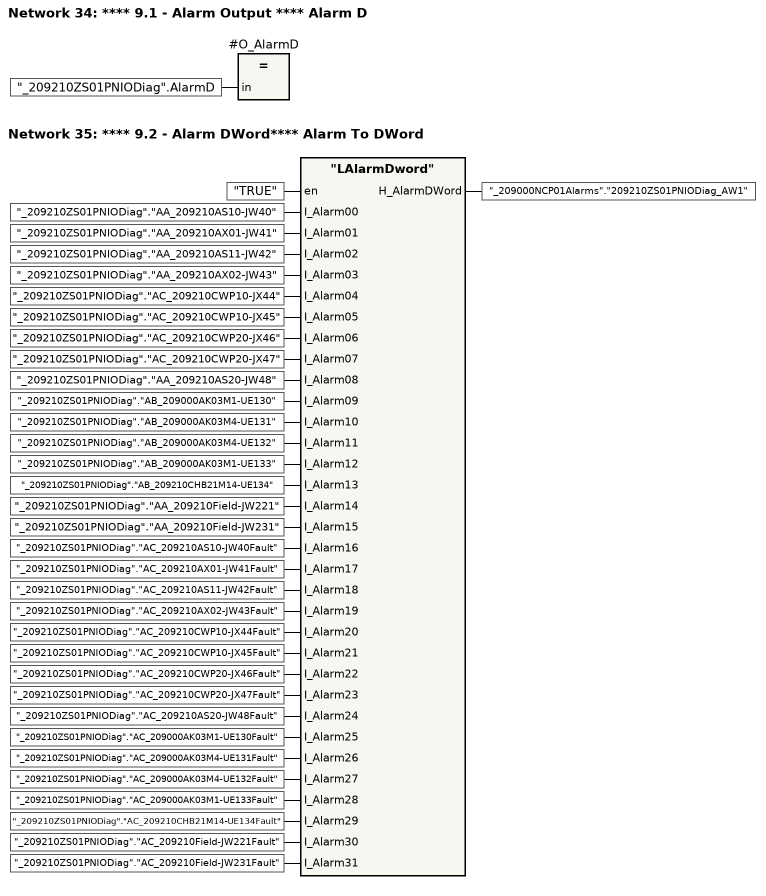
   #O_AlarmD := "_209210ZS01PNIODiag".AlarmD;
END_REGION

REGION Network 35: **** 9.2 - Alarm DWord**** Alarm To DWord
   // Alarm Word
   IF "TRUE" THEN
       "LAlarmDword"(I_Alarm00 := "_209210ZS01PNIODiag"."AA_209210AS10-JW40",
                     I_Alarm01 := "_209210ZS01PNIODiag"."AA_209210AX01-JW41",
                     I_Alarm02 := "_209210ZS01PNIODiag"."AA_209210AS11-JW42",
                     I_Alarm03 := "_209210ZS01PNIODiag"."AA_209210AX02-JW43",
                     I_Alarm04 := "_209210ZS01PNIODiag"."AC_209210CWP10-JX44",
                     I_Alarm05 := "_209210ZS01PNIODiag"."AC_209210CWP10-JX45",
                     I_Alarm06 := "_209210ZS01PNIODiag"."AC_209210CWP20-JX46",
                     I_Alarm07 := "_209210ZS01PNIODiag"."AC_209210CWP20-JX47",
                     I_Alarm08 := "_209210ZS01PNIODiag"."AA_209210AS20-JW48",
                     I_Alarm09 := "_209210ZS01PNIODiag"."AB_209000AK03M1-UE130",
                     I_Alarm10 := "_209210ZS01PNIODiag"."AB_209000AK03M4-UE131",
                     I_Alarm11 := "_209210ZS01PNIODiag"."AB_209000AK03M4-UE132",
                     I_Alarm12 := "_209210ZS01PNIODiag"."AB_209000AK03M1-UE133",
                     I_Alarm13 := "_209210ZS01PNIODiag"."AB_209210CHB21M14-UE134",
                     I_Alarm14 := "_209210ZS01PNIODiag"."AA_209210Field-JW221",
                     I_Alarm15 := "_209210ZS01PNIODiag"."AA_209210Field-JW231",
                     I_Alarm16 := "_209210ZS01PNIODiag"."AC_209210AS10-JW40Fault",
                     I_Alarm17 := "_209210ZS01PNIODiag"."AC_209210AX01-JW41Fault",
                     I_Alarm18 := "_209210ZS01PNIODiag"."AC_209210AS11-JW42Fault",
                     I_Alarm19 := "_209210ZS01PNIODiag"."AC_209210AX02-JW43Fault",
                     I_Alarm20 := "_209210ZS01PNIODiag"."AC_209210CWP10-JX44Fault",
                     I_Alarm21 := "_209210ZS01PNIODiag"."AC_209210CWP10-JX45Fault",
                     I_Alarm22 := "_209210ZS01PNIODiag"."AC_209210CWP20-JX46Fault",
                     I_Alarm23 := "_209210ZS01PNIODiag"."AC_209210CWP20-JX47Fault",
                     I_Alarm24 := "_209210ZS01PNIODiag"."AC_209210AS20-JW48Fault",
                     I_Alarm25 := "_209210ZS01PNIODiag"."AC_209000AK03M1-UE130Fault",
                     I_Alarm26 := "_209210ZS01PNIODiag"."AC_209000AK03M4-UE131Fault",
                     I_Alarm27 := "_209210ZS01PNIODiag"."AC_209000AK03M4-UE132Fault",
                     I_Alarm28 := "_209210ZS01PNIODiag"."AC_209000AK03M1-UE133Fault",
                     I_Alarm29 := "_209210ZS01PNIODiag"."AC_209210CHB21M14-UE134Fault",
                     I_Alarm30 := "_209210ZS01PNIODiag"."AC_209210Field-JW221Fault",
                     I_Alarm31 := "_209210ZS01PNIODiag"."AC_209210Field-JW231Fault",
                     H_AlarmDWord => "_209000NCP01Alarms"."209210ZS01PNIODiag_AW1");
   END_IF;
END_REGION
END_FUNCTION
